FUNCTION_BLOCK FB_do
VAR_INPUT
END_VAR
VAR_OUTPUT
END_VAR
VAR
END_VAR

END_FUNCTION_BLOCK

(* stored: Version 1.1.0.1, ProductVersion 3.1.4024.12
   POU FB_do: Id {6749007b-e9a2-496a-a70b-1cf05b2d5b2c}, SpecialFunc None *)
